PROGRAM main
VAR
	SW1 AT %IX0.0 : bool;
	SW2 AT %IX0.1 : bool;
	SW3 AT %IX0.2 : bool;
	Master_Stop AT %IX0.3 : bool;
	Lamp AT %QX0.0 : bool;
END_VAR

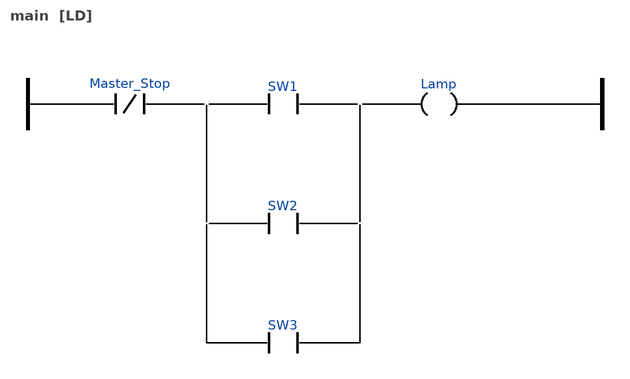
(* LD diagram, written out as Structured Text *)
Lamp := NOT Master_Stop AND (SW1 OR SW2 OR SW3);
END_PROGRAM
